(* IEC 61131-3 sources: Industry-PLC-LLM/data/PLCBEAD_repo/PLCBEAD_PLCEmbed-main/PLC-BEAD/Source/GEB/FF_D2E, 1 file *)

(* ---- FF_D2E.ST ---- *)
FUNCTION_BLOCK FF_D2E
	VAR_INPUT
		D0 :	BOOL;
		D1 :	BOOL;
		CLK :	BOOL;
		RST :	BOOL;
	END_VAR

	VAR_OUTPUT
		Q0 :	BOOL;
		Q1 :	BOOL;
	END_VAR

	VAR
		edge :	BOOL;
	END_VAR

	IF RST THEN
		Q0 := FALSE;
		Q1 := FALSE;
	ELSIF CLK AND NOT edge THEN
		Q0 := D0;
		Q1 := D1;
	END_IF;
	edge := CLK;

END_FUNCTION_BLOCK

PROGRAM program0
  VAR
	D0  :	BOOL;
	D1  :	BOOL;
	CLK :	BOOL;
	RST :	BOOL;

	Q0 :	BOOL;
	Q1 :	BOOL;

	func_block : FF_D2E;
  END_VAR
	func_block.D0  :=D0 ;
	func_block.D1  :=D1 ;
	func_block.CLK :=CLK;
	func_block.RST :=RST;
	func_block();
	Q0 := func_block.Q0;
	Q1 := func_block.Q1;
END_PROGRAM
